PROGRAM MAIN
VAR
	fbBlinker : FB_Blinker;
	fbCaseBlinker : FB_CaseBlinker;
	
	bIsStartPressed : BOOL;
	bIsCaseStartPressed : BOOL;
	
	dwTimeOn : DWORD := 2000;
	dwTimeOff : DWORD := 1000;
	dwCaseTimeOn : DWORD := 2000;
	dwCaseTimeOff : DWORD := 1000;
END_VAR

fbBlinker(bIsStartPressed := bIsStartPressed, dwTimeOn := dwTimeOn, dwTimeOff := dwTimeOff);

fbCaseBlinker(bIsStartPressed := bIsCaseStartPressed, dwTimeOn := dwCaseTimeOn, dwTimeOff := dwCaseTimeOff);

fbCaseBlinker(dwTimeOn := dwCaseTimeOn, dwTimeOff := dwCaseTimeOff);

END_PROGRAM

(* stored: Version 1.1.0.1, ProductVersion 3.1.4024.12
   POU MAIN: Id {123b3537-2b46-43a3-a8d2-3b8e902ef314}, SpecialFunc None *)
